{attribute 'qualified_only'}
VAR_GLOBAL
	bGlobalReset : bool := false ;  
END_VAR

(* stored: Version 1.1.0.1, ProductVersion 3.1.4024.12
   GVL GVL: Id {632c5b18-c91c-4915-aa02-81171c2efa54} *)
